(* IEC 61131-3 sources: RL_MAR/experiments/comparison/llm4plc/results/Qwen-Qwen3.5-9B_20260506_150728/20260506_162334, 4 files *)

(* ---- generated_code_iteration_0.st ---- *)
START_ST
TYPE T_GARAGE_SLOT:
STRUCT
Occupied : BOOL;
VehicleNumber : INT;
END_STRUCT;
END_TYPE

TYPE T_TRUCK_INFO:
STRUCT
row : INT;
col : INT;
VehicleNumber : INT;
END_STRUCT;
END_TYPE

FUNCTION_BLOCK TruckGarage
VAR_INPUT
enter_flag : BOOL;
exit_flag : BOOL;
VehicleNumber_in : INT;
END_VAR
VAR_OUTPUT
truck : T_TRUCK_INFO;
END_VAR
VAR_IN_OUT
garage : ARRAY[1..3, 1..5] OF T_GARAGE_SLOT;
END_VAR
VAR
CurrentState : INT;
PreviousState : INT;
FoundSlot : BOOL;
SearchRow : INT;
SearchCol : INT;
ExitFound : BOOL;
i : INT;
j : INT;
END_VAR

// --- STATE MACHINE LOGIC ---
// Initialize state if this is the first execution or reset
IF CurrentState = 0 AND PreviousState <> 0 THEN
    CurrentState := 0;
    PreviousState := 0;
    truck.row := 0;
    truck.col := 0;
    truck.VehicleNumber := 0;
    FoundSlot := FALSE;
    ExitFound := FALSE;
END_IF

// State 0: IDLE (Waiting for a request)
IF CurrentState = 0 THEN
    PreviousState := 0;

    // Transition to ENTRY_PROCESSING
    IF enter_flag = TRUE THEN
        CurrentState := 1;
        FoundSlot := FALSE;
    END_IF;

    // Transition to EXIT_PROCESSING
    IF exit_flag = TRUE THEN
        CurrentState := 2;
        ExitFound := FALSE;
    END_IF;

    // Reset output if no action is taken
    IF enter_flag = FALSE AND exit_flag = FALSE THEN
        truck.row := 0;
        truck.col := 0;
        truck.VehicleNumber := 0;
    END_IF;
END_IF;

// State 1: ENTRY_PROCESSING (Search and Allocate)
IF CurrentState = 1 THEN
    PreviousState := 1;
    FoundSlot := FALSE;
    SearchRow := 0;
    SearchCol := 0;

    // Iterate rows from 3 down to 1 (Latter Row First)
    FOR i := 3 DOWNTO 1 DO
        // Iterate columns from 5 down to 1 (Latter Column First)
        FOR j := 5 DOWNTO 1 DO
            IF garage[i, j].Occupied = FALSE THEN
                // Slot found
                garage[i, j].Occupied := TRUE;
                garage[i, j].VehicleNumber := VehicleNumber_in;
                FoundSlot := TRUE;
                SearchRow := i;
                SearchCol := j;
                EXIT; // Exit inner loop
            END_IF;
        END_FOR;
        IF FoundSlot = TRUE THEN
            EXIT; // Exit outer loop
        END_IF;
    END_FOR;

    // Update output and transition to COMPLETED
    IF FoundSlot = TRUE THEN
        truck.row := SearchRow;
        truck.col := SearchCol;
        truck.VehicleNumber := VehicleNumber_in;
        CurrentState := 3;
    END_IF;
END_IF;

// State 2: EXIT_PROCESSING (Search and Release)
IF CurrentState = 2 THEN
    PreviousState := 2;
    ExitFound := FALSE;
    SearchRow := 0;
    SearchCol := 0;

    // Iterate rows from 1 up to 3 (Former Row First)
    FOR i := 1 TO 3 DO
        // Iterate columns from 1 up to 5 (Former Column First)
        FOR j := 1 TO 5 DO
            IF garage[i, j].Occupied = TRUE AND garage[i, j].VehicleNumber = VehicleNumber_in THEN
                // Truck found
                garage[i, j].Occupied := FALSE;
                garage[i, j].VehicleNumber := 0;
                ExitFound := TRUE;
                SearchRow := i;
                SearchCol := j;
                EXIT; // Exit inner loop
            END_IF;
        END_FOR;
        IF ExitFound = TRUE THEN
            EXIT; // Exit outer loop
        END_IF;
    END_FOR;

    // Update output and transition to COMPLETED
    IF ExitFound = TRUE THEN
        truck.row := SearchRow;
        truck.col := SearchCol;
        truck.VehicleNumber := VehicleNumber_in;
        CurrentState := 3;
    END_IF;
END_IF;

// State 3: COMPLETED (Request handled, return to IDLE)
IF CurrentState = 3 THEN
    PreviousState := 3;
    // State remains 3 until the next PLC cycle starts, effectively holding the result
    // The transition back to 0 happens at the beginning of the next scan
END_IF;

END_FUNCTION_BLOCK
END_ST

(* ---- generated_code_iteration_1.st ---- *)
START_REASON
The validation feedback indicates a "Unknown type: 'T_TRUCK_INFO'" error. In IEC 61131-3 Structured Text (ST), specifically within the CODESYS compiler environment, type definitions (TYPE ... END_TYPE) must be placed at the global scope (outside of any FUNCTION_BLOCK, PROGRAM, or FUNCTION) before they are referenced.

In the provided code, `TYPE T_TRUCK_INFO` is defined inside the `FUNCTION_BLOCK TruckGarage`. This is syntactically incorrect. The compiler encounters the reference to `T_TRUCK_INFO` in the `VAR_OUTPUT` section before it has finished parsing the block, or simply because local type definitions are not allowed in this context.

To fix this:
1.  Move the `TYPE T_GARAGE_SLOT` and `TYPE T_TRUCK_INFO` definitions to the very top of the code, outside the `FUNCTION_BLOCK`.
2.  Ensure the `FUNCTION_BLOCK` uses these globally defined types.
3.  Maintain the `FUNCTION_BLOCK` structure as required.
4.  Ensure all variable sections use `END_VAR` correctly.
START_END
END_REASON

START_ST
TYPE T_GARAGE_SLOT:
STRUCT
Occupied : BOOL;
VehicleNumber : INT;
END_STRUCT;
END_TYPE

TYPE T_TRUCK_INFO:
STRUCT
row : INT;
col : INT;
VehicleNumber : INT;
END_STRUCT;
END_TYPE

FUNCTION_BLOCK TruckGarage
VAR_INPUT
enter_flag : BOOL;
exit_flag : BOOL;
VehicleNumber_in : INT;
END_VAR
VAR_OUTPUT
truck : T_TRUCK_INFO;
END_VAR
VAR_IN_OUT
garage : ARRAY[1..3, 1..5] OF T_GARAGE_SLOT;
END_VAR
VAR
CurrentState : INT;
PreviousState : INT;
FoundSlot : BOOL;
SearchRow : INT;
SearchCol : INT;
ExitFound : BOOL;
i : INT;
j : INT;
END_VAR

// --- STATE MACHINE LOGIC ---
// Initialize state if this is the first execution or reset
IF CurrentState = 0 AND PreviousState <> 0 THEN
    CurrentState := 0;
    PreviousState := 0;
    truck.row := 0;
    truck.col := 0;
    truck.VehicleNumber := 0;
    FoundSlot := FALSE;
    ExitFound := FALSE;
END_IF

// State 0: IDLE (Waiting for a request)
IF CurrentState = 0 THEN
    PreviousState := 0;

    // Transition to ENTRY_PROCESSING
    IF enter_flag = TRUE THEN
        CurrentState := 1;
        FoundSlot := FALSE;
    END_IF;

    // Transition to EXIT_PROCESSING
    IF exit_flag = TRUE THEN
        CurrentState := 2;
        ExitFound := FALSE;
    END_IF;

    // Reset output if no action is taken
    IF enter_flag = FALSE AND exit_flag = FALSE THEN
        truck.row := 0;
        truck.col := 0;
        truck.VehicleNumber := 0;
    END_IF;
END_IF;

// State 1: ENTRY_PROCESSING (Search and Allocate)
IF CurrentState = 1 THEN
    PreviousState := 1;
    FoundSlot := FALSE;
    SearchRow := 0;
    SearchCol := 0;

    // Iterate rows from 3 down to 1 (Latter Row First)
    FOR i := 3 DOWNTO 1 DO
        // Iterate columns from 5 down to 1 (Latter Column First)
        FOR j := 5 DOWNTO 1 DO
            IF garage[i, j].Occupied = FALSE THEN
                // Slot found
                garage[i, j].Occupied := TRUE;
                garage[i, j].VehicleNumber := VehicleNumber_in;
                FoundSlot := TRUE;
                SearchRow := i;
                SearchCol := j;
                EXIT; // Exit inner loop
            END_IF;
        END_FOR;
        IF FoundSlot = TRUE THEN
            EXIT; // Exit outer loop
        END_IF;
    END_FOR;

    // Update output and transition to COMPLETED
    IF FoundSlot = TRUE THEN
        truck.row := SearchRow;
        truck.col := SearchCol;
        truck.VehicleNumber := VehicleNumber_in;
        CurrentState := 3;
    END_IF;
END_IF;

// State 2: EXIT_PROCESSING (Search and Release)
IF CurrentState = 2 THEN
    PreviousState := 2;
    ExitFound := FALSE;
    SearchRow := 0;
    SearchCol := 0;

    // Iterate rows from 1 up to 3 (Former Row First)
    FOR i := 1 TO 3 DO
        // Iterate columns from 1 up to 5 (Former Column First)
        FOR j := 1 TO 5 DO
            IF garage[i, j].Occupied = TRUE AND garage[i, j].VehicleNumber = VehicleNumber_in THEN
                // Truck found
                garage[i, j].Occupied := FALSE;
                garage[i, j].VehicleNumber := 0;
                ExitFound := TRUE;
                SearchRow := i;
                SearchCol := j;
                EXIT; // Exit inner loop
            END_IF;
        END_FOR;
        IF ExitFound = TRUE THEN
            EXIT; // Exit outer loop
        END_IF;
    END_FOR;

    // Update output and transition to COMPLETED
    IF ExitFound = TRUE THEN
        truck.row := SearchRow;
        truck.col := SearchCol;
        truck.VehicleNumber := VehicleNumber_in;
        CurrentState := 3;
    END_IF;
END_IF;

// State 3: COMPLETED (Request handled, return to IDLE)
IF CurrentState = 3 THEN
    PreviousState := 3;
    // State remains 3 until the next PLC cycle starts, effectively holding the result
    // The transition back to 0 happens at the beginning of the next scan
END_IF;

END_FUNCTION_BLOCK
END_ST

(* ---- generated_code_iteration_2.st ---- *)
START_REASON
The previous attempt failed because the `TYPE` definitions (`T_GARAGE_SLOT` and `T_TRUCK_INFO`) were placed **inside** the `FUNCTION_BLOCK TruckGarage`. In IEC 61131-3 (and specifically in CODESYS), type definitions must be declared at the **global scope**, outside of any program, function block, or function.

The compiler error "Unknown type: 'T_TRUCK_INFO'" occurs because when the compiler parses the `VAR_OUTPUT` section of the function block, it looks for the definition of `T_TRUCK_INFO`. Since the definition is nested inside the function block (which hasn't finished parsing yet), the compiler cannot resolve the type.

To fix this:
1.  Move the `TYPE T_GARAGE_SLOT` and `TYPE T_TRUCK_INFO` definitions to the very top of the code, before the `FUNCTION_BLOCK` declaration.
2.  Ensure the `FUNCTION_BLOCK` references these globally defined types.
3.  Maintain the `FUNCTION_BLOCK` structure and logic as originally intended.
4.  Ensure all variable sections strictly use `END_VAR`.
END_REASON

START_ST
TYPE T_GARAGE_SLOT
STRUCT
    Occupied : BOOL;
    VehicleNumber : INT;
END_STRUCT
END_TYPE

TYPE T_TRUCK_INFO
STRUCT
    row : INT;
    col : INT;
    VehicleNumber : INT;
END_STRUCT
END_TYPE

FUNCTION_BLOCK TruckGarage
VAR_INPUT
    enter_flag : BOOL;
    exit_flag : BOOL;
    VehicleNumber_in : INT;
END_VAR

VAR_OUTPUT
    truck : T_TRUCK_INFO;
END_VAR

VAR_IN_OUT
    garage : ARRAY[1..3, 1..5] OF T_GARAGE_SLOT;
END_VAR

VAR
    CurrentState : INT;
    PreviousState : INT;
    FoundSlot : BOOL;
    SearchRow : INT;
    SearchCol : INT;
    ExitFound : BOOL;
    i : INT;
    j : INT;
END_VAR

// --- STATE MACHINE LOGIC ---
// Initialize state if this is the first execution or reset
IF CurrentState = 0 AND PreviousState <> 0 THEN
    CurrentState := 0;
    PreviousState := 0;
    truck.row := 0;
    truck.col := 0;
    truck.VehicleNumber := 0;
    FoundSlot := FALSE;
    ExitFound := FALSE;
END_IF

// State 0: IDLE (Waiting for a request)
IF CurrentState = 0 THEN
    PreviousState := 0;

    // Transition to ENTRY_PROCESSING
    IF enter_flag = TRUE THEN
        CurrentState := 1;
        FoundSlot := FALSE;
    END_IF;

    // Transition to EXIT_PROCESSING
    IF exit_flag = TRUE THEN
        CurrentState := 2;
        ExitFound := FALSE;
    END_IF;

    // Reset output if no action is taken
    IF enter_flag = FALSE AND exit_flag = FALSE THEN
        truck.row := 0;
        truck.col := 0;
        truck.VehicleNumber := 0;
    END_IF;
END_IF;

// State 1: ENTRY_PROCESSING (Search and Allocate)
IF CurrentState = 1 THEN
    PreviousState := 1;
    FoundSlot := FALSE;
    SearchRow := 0;
    SearchCol := 0;

    // Iterate rows from 3 down to 1 (Latter Row First)
    FOR i := 3 DOWNTO 1 DO
        // Iterate columns from 5 down to 1 (Latter Column First)
        FOR j := 5 DOWNTO 1 DO
            IF garage[i, j].Occupied = FALSE THEN
                // Slot found
                garage[i, j].Occupied := TRUE;
                garage[i, j].VehicleNumber := VehicleNumber_in;
                FoundSlot := TRUE;
                SearchRow := i;
                SearchCol := j;
                EXIT; // Exit inner loop
            END_IF;
        END_FOR;
        IF FoundSlot = TRUE THEN
            EXIT; // Exit outer loop
        END_IF;
    END_FOR;

    // Update output and transition to COMPLETED
    IF FoundSlot = TRUE THEN
        truck.row := SearchRow;
        truck.col := SearchCol;
        truck.VehicleNumber := VehicleNumber_in;
        CurrentState := 3;
    END_IF;
END_IF;

// State 2: EXIT_PROCESSING (Search and Release)
IF CurrentState = 2 THEN
    PreviousState := 2;
    ExitFound := FALSE;
    SearchRow := 0;
    SearchCol := 0;

    // Iterate rows from 1 up to 3 (Former Row First)
    FOR i := 1 TO 3 DO
        // Iterate columns from 1 up to 5 (Former Column First)
        FOR j := 1 TO 5 DO
            IF garage[i, j].Occupied = TRUE AND garage[i, j].VehicleNumber = VehicleNumber_in THEN
                // Truck found
                garage[i, j].Occupied := FALSE;
                garage[i, j].VehicleNumber := 0;
                ExitFound := TRUE;
                SearchRow := i;
                SearchCol := j;
                EXIT; // Exit inner loop
            END_IF;
        END_FOR;
        IF ExitFound = TRUE THEN
            EXIT; // Exit outer loop
        END_IF;
    END_FOR;

    // Update output and transition to COMPLETED
    IF ExitFound = TRUE THEN
        truck.row := SearchRow;
        truck.col := SearchCol;
        truck.VehicleNumber := VehicleNumber_in;
        CurrentState := 3;
    END_IF;
END_IF;

// State 3: COMPLETED (Request handled, return to IDLE)
IF CurrentState = 3 THEN
    PreviousState := 3;
    // State remains 3 until the next PLC cycle starts, effectively holding the result
    // The transition back to 0 happens at the beginning of the next scan
END_IF;

END_FUNCTION_BLOCK
END_ST

(* ---- generated_code_iteration_3.st ---- *)
START_REASON
The previous attempt failed because the `FUNCTION_BLOCK` definition was placed **before** the `TYPE` definitions in the source code. In IEC 61131-3 (and specifically in CODESYS), while types can technically be defined globally, the compiler requires that all types used within a program block (like `FUNCTION_BLOCK`) must be declared **before** the block that uses them.

In the previous code:
1. `FUNCTION_BLOCK TruckGarage` was declared first.
2. Inside `VAR_OUTPUT`, the type `T_TRUCK_INFO` was referenced.
3. The definition of `TYPE T_TRUCK_INFO` appeared **after** the `FUNCTION_BLOCK` declaration.

When the compiler parses the `FUNCTION_BLOCK`, it encounters the reference to `T_TRUCK_INFO` before it has seen the definition, resulting in the error "Unknown type: 'T_TRUCK_INFO'".

To fix this:
1. Move the `TYPE T_GARAGE_SLOT` and `TYPE T_TRUCK_INFO` definitions to the very top of the file.
2. Ensure the `FUNCTION_BLOCK` declaration comes **after** these type definitions.
3. Maintain the `FUNCTION_BLOCK` structure and logic exactly as intended.
4. Ensure all variable sections strictly use `END_VAR`.
END_REASON

START_ST
TYPE T_GARAGE_SLOT
STRUCT
    Occupied : BOOL;
    VehicleNumber : INT;
END_STRUCT
END_TYPE

TYPE T_TRUCK_INFO
STRUCT
    row : INT;
    col : INT;
    VehicleNumber : INT;
END_STRUCT
END_TYPE

FUNCTION_BLOCK TruckGarage
VAR_INPUT
    enter_flag : BOOL;
    exit_flag : BOOL;
    VehicleNumber_in : INT;
END_VAR

VAR_OUTPUT
    truck : T_TRUCK_INFO;
END_VAR

VAR_IN_OUT
    garage : ARRAY[1..3, 1..5] OF T_GARAGE_SLOT;
END_VAR

VAR
    CurrentState : INT;
    PreviousState : INT;
    FoundSlot : BOOL;
    SearchRow : INT;
    SearchCol : INT;
    ExitFound : BOOL;
    i : INT;
    j : INT;
END_VAR

// --- STATE MACHINE LOGIC ---
// Initialize state if this is the first execution or reset
IF CurrentState = 0 AND PreviousState <> 0 THEN
    CurrentState := 0;
    PreviousState := 0;
    truck.row := 0;
    truck.col := 0;
    truck.VehicleNumber := 0;
    FoundSlot := FALSE;
    ExitFound := FALSE;
END_IF

// State 0: IDLE (Waiting for a request)
IF CurrentState = 0 THEN
    PreviousState := 0;

    // Transition to ENTRY_PROCESSING
    IF enter_flag = TRUE THEN
        CurrentState := 1;
        FoundSlot := FALSE;
    END_IF;

    // Transition to EXIT_PROCESSING
    IF exit_flag = TRUE THEN
        CurrentState := 2;
        ExitFound := FALSE;
    END_IF;

    // Reset output if no action is taken
    IF enter_flag = FALSE AND exit_flag = FALSE THEN
        truck.row := 0;
        truck.col := 0;
        truck.VehicleNumber := 0;
    END_IF;
END_IF;

// State 1: ENTRY_PROCESSING (Search and Allocate)
IF CurrentState = 1 THEN
    PreviousState := 1;
    FoundSlot := FALSE;
    SearchRow := 0;
    SearchCol := 0;

    // Iterate rows from 3 down to 1 (Latter Row First)
    FOR i := 3 DOWNTO 1 DO
        // Iterate columns from 5 down to 1 (Latter Column First)
        FOR j := 5 DOWNTO 1 DO
            IF garage[i, j].Occupied = FALSE THEN
                // Slot found
                garage[i, j].Occupied := TRUE;
                garage[i, j].VehicleNumber := VehicleNumber_in;
                FoundSlot := TRUE;
                SearchRow := i;
                SearchCol := j;
                EXIT; // Exit inner loop
            END_IF;
        END_FOR;
        IF FoundSlot = TRUE THEN
            EXIT; // Exit outer loop
        END_IF;
    END_FOR;

    // Update output and transition to COMPLETED
    IF FoundSlot = TRUE THEN
        truck.row := SearchRow;
        truck.col := SearchCol;
        truck.VehicleNumber := VehicleNumber_in;
        CurrentState := 3;
    END_IF;
END_IF;

// State 2: EXIT_PROCESSING (Search and Release)
IF CurrentState = 2 THEN
    PreviousState := 2;
    ExitFound := FALSE;
    SearchRow := 0;
    SearchCol := 0;

    // Iterate rows from 1 up to 3 (Former Row First)
    FOR i := 1 TO 3 DO
        // Iterate columns from 1 up to 5 (Former Column First)
        FOR j := 1 TO 5 DO
            IF garage[i, j].Occupied = TRUE AND garage[i, j].VehicleNumber = VehicleNumber_in THEN
                // Truck found
                garage[i, j].Occupied := FALSE;
                garage[i, j].VehicleNumber := 0;
                ExitFound := TRUE;
                SearchRow := i;
                SearchCol := j;
                EXIT; // Exit inner loop
            END_IF;
        END_FOR;
        IF ExitFound = TRUE THEN
            EXIT; // Exit outer loop
        END_IF;
    END_FOR;

    // Update output and transition to COMPLETED
    IF ExitFound = TRUE THEN
        truck.row := SearchRow;
        truck.col := SearchCol;
        truck.VehicleNumber := VehicleNumber_in;
        CurrentState := 3;
    END_IF;
END_IF;

// State 3: COMPLETED (Request handled, return to IDLE)
IF CurrentState = 3 THEN
    PreviousState := 3;
    // State remains 3 until the next PLC cycle starts, effectively holding the result
    // The transition back to 0 happens at the beginning of the next scan
END_IF;

END_FUNCTION_BLOCK
END_ST
